// SIMATIC S7-200 project (STEP 7-Micro/WIN), CPU 221 REL 01.10

SYMBOL_TABLE USER1
phim_2           I0.0
phim_4           I0.1
phim_6           I0.2
clear            I0.3
start            I0.4
stopp            I0.5
den              Q0.0
END_SYMBOL_TABLE

ORGANIZATION_BLOCK MAIN:OB1
TITLE=PROGRAM COMMENTS
BEGIN
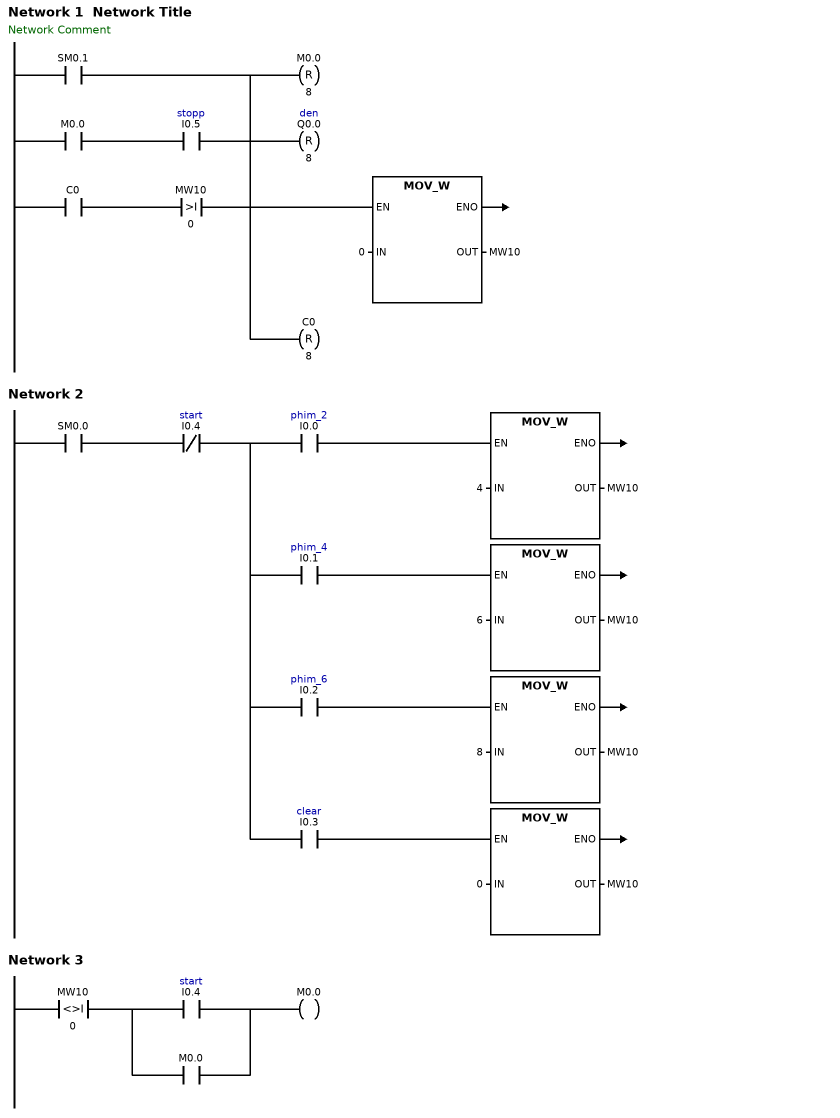
Network 1 // Network Title
// Network Comment
LD     SM0.1
LD     M0.0
A      stopp:I0.5
OLD
LD     C0
AW>    MW10, 0
OLD
R      M0.0, 8
R      den:Q0.0, 8
MOVW   0, MW10
R      C0, 8
Network 2
LD     SM0.0
AN     start:I0.4
LPS
A      phim_2:I0.0
MOVW   4, MW10
LRD
A      phim_4:I0.1
MOVW   6, MW10
LRD
A      phim_6:I0.2
MOVW   8, MW10
LPP
A      clear:I0.3
MOVW   0, MW10
Network 3
LDW<>  MW10, 0
LD     start:I0.4
O      M0.0
ALD
=      M0.0
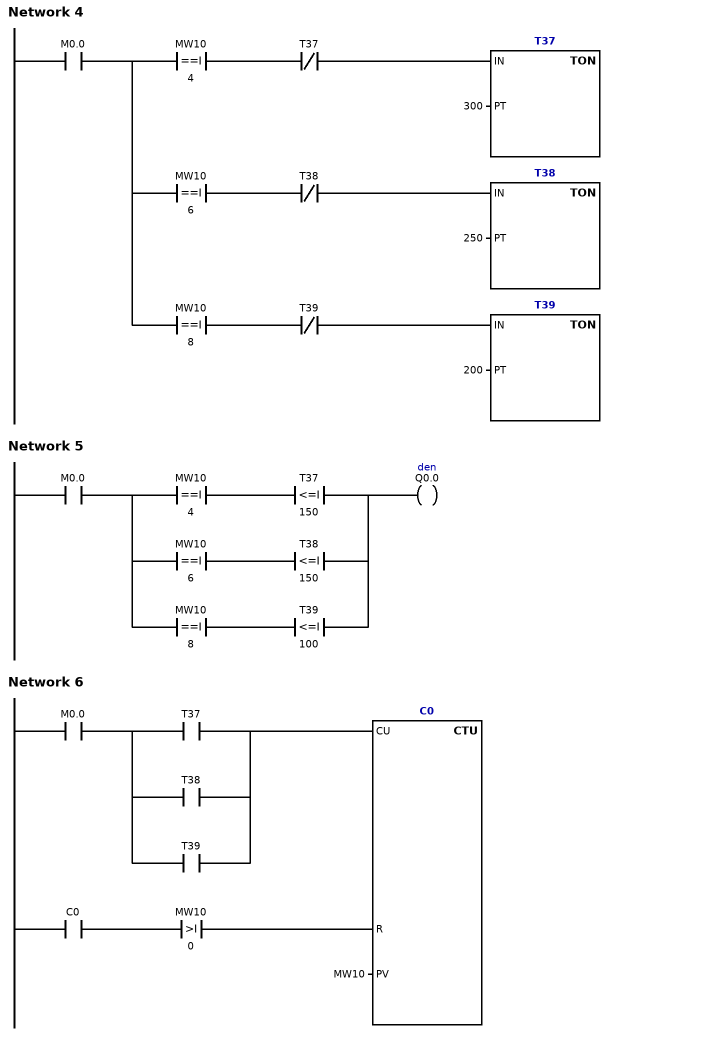
Network 4
LD     M0.0
LPS
AW=    MW10, 4
AN     T37
TON    T37, 300
LRD
AW=    MW10, 6
AN     T38
TON    T38, 250
LPP
AW=    MW10, 8
AN     T39
TON    T39, 200
Network 5
LD     M0.0
LDW=   MW10, 4
AW<=   T37, 150
LDW=   MW10, 6
AW<=   T38, 150
OLD
LDW=   MW10, 8
AW<=   T39, 100
OLD
ALD
=      den:Q0.0
Network 6
LD     M0.0
LD     T37
O      T38
O      T39
ALD
LD     C0
AW>    MW10, 0
CTU    C0, MW10
END_ORGANIZATION_BLOCK
